{attribute 'GeneratedUsingTerminal: EK1100-0000-0018'}
{attribute addProperty BoxType "EK1100-0000-0018"}
{attribute addProperty Id "Beckhoff_EM7xxxEK1122Beckhoff_EM7xxxEK1122_DEE9974A2A_0001_EM7004_0000_9995EM7004_C205438B84A_0002_EM7004_0000_9996EM7004_7C77157F107A_0003_EM7004_0000_9997EM7004_7C77157F107A_0004_EM7004_0000_0016EM7004_7D59F373111A_0005_EM7004_0000_0017EM7004_91F96046111A_0006_EM7004_0000_0018EM7004_91F96046111"}
{attribute addProperty CRC "427920810"}
{attribute addProperty Size "633"}
TYPE Beckhoff_EM7xxx_19818DAA EXTENDS EK1100_1FC0878B :
STRUCT
	{attribute addProperty Name "Beckhoff_EM7xxxEK1122"}
	{attribute addProperty PreviousPort "Beckhoff EM7xxx : B"}
	Beckhoff_EM7xxxEK1122 : Beckhoff_EM7xxxEK1122_DEE9974A;
	{attribute addProperty Name "A_0001_EM7004_0000_9995"}
	{attribute addProperty PreviousPort "Beckhoff EM7xxxEK1122 : C"}
	A_0001_EM7004_0000_9995 : EM7004_C205438B;
	{attribute addProperty Name "A_0002_EM7004_0000_9996"}
	{attribute addProperty PreviousPort "A_0001(EM7004-0000-9995) : B"}
	A_0002_EM7004_0000_9996 : EM7004_7C77157F;
	{attribute addProperty Name "A_0003_EM7004_0000_9997"}
	{attribute addProperty PreviousPort "A_0002(EM7004-0000-9996) : B"}
	A_0003_EM7004_0000_9997 : EM7004_7C77157F;
	{attribute addProperty Name "A_0004_EM7004_0000_0016"}
	{attribute addProperty PreviousPort "A_0003(EM7004-0000-9997) : B"}
	A_0004_EM7004_0000_0016 : EM7004_7D59F373;
	{attribute addProperty Name "A_0005_EM7004_0000_0017"}
	{attribute addProperty PreviousPort "A_0004(EM7004-0000-0016) : B"}
	A_0005_EM7004_0000_0017 : EM7004_91F96046;
	{attribute addProperty Name "A_0006_EM7004_0000_0018"}
	{attribute addProperty PreviousPort "A_0005(EM7004-0000-0017) : B"}
	A_0006_EM7004_0000_0018 : EM7004_91F96046;
END_STRUCT
END_TYPE

(* stored: Version 1.2.0.0, ProductVersion 3.1.4024.9
   DUT Beckhoff_EM7xxx_19818DAA: Id {d3c2b238-5257-4449-b214-a86a5cdc2d8a} *)
